Yaskawa INFORM job: AAA.JBI

/JOB
//NAME AAA
//POS
///NPOS 204,0,0,0,0,0
///TOOL 11
///POSTYPE PULSE
///PULSE
C00000=-67760,-23601,-34425,-10736,-67084,75715
C00001=-67760,-23601,-34425,-10736,-67084,75715
C00002=-69499,-30257,-42570,-18909,-69402,74527
C00003=-69664,-30877,-43349,-19628,-69583,74428
C00004=-69705,-31406,-44012,-20162,-69808,74223
C00005=-69657,-31867,-44586,-20565,-70063,73943
C00006=-69549,-32276,-45094,-20883,-70341,73613
C00007=-69400,-32646,-45556,-21151,-70634,73252
C00008=-69228,-32989,-45983,-21392,-70939,72872
C00009=-69041,-33312,-46388,-21624,-71251,72483
C00010=-68847,-33623,-46778,-21857,-71568,72091
C00011=-68651,-33924,-47158,-22097,-71886,71699
C00012=-68455,-34220,-47531,-22349,-72206,71309
C00013=-68258,-34512,-47898,-22611,-72524,70923
C00014=-68061,-34801,-48261,-22885,-72842,70541
C00015=-67864,-35088,-48619,-23168,-73158,70162
C00016=-67664,-35372,-48972,-23459,-73473,69786
C00017=-67462,-35653,-49319,-23757,-73786,69413
C00018=-67255,-35930,-49660,-24059,-74096,69042
C00019=-67043,-36203,-49993,-24363,-74405,68672
C00020=-66826,-36471,-50319,-24671,-74712,68304
C00021=-66603,-36736,-50637,-24979,-75016,67938
C00022=-66373,-36997,-50948,-25288,-75318,67573
C00023=-66137,-37255,-51251,-25599,-75616,67211
C00024=-65895,-37511,-51549,-25910,-75911,66851
C00025=-65647,-37765,-51840,-26222,-76201,66493
C00026=-65393,-38019,-52126,-26535,-76486,66139
C00027=-65133,-38273,-52409,-26849,-76767,65789
C00028=-64867,-38529,-52687,-27164,-77041,65442
C00029=-64596,-38787,-52963,-27481,-77309,65099
C00030=-64319,-39049,-53236,-27798,-77570,64761
C00031=-64036,-39314,-53506,-28117,-77824,64427
C00032=-63747,-39584,-53775,-28435,-78070,64097
C00033=-63453,-39857,-54041,-28754,-78309,63772
C00034=-63152,-40136,-54305,-29073,-78541,63450
C00035=-62844,-40418,-54566,-29390,-78765,63132
C00036=-62529,-40703,-54824,-29706,-78981,62818
C00037=-62206,-40991,-55077,-30019,-79190,62508
C00038=-61875,-41281,-55326,-30328,-79393,62200
C00039=-61536,-41572,-55568,-30634,-79589,61896
C00040=-61188,-41863,-55804,-30936,-79778,61593
C00041=-60831,-42153,-56033,-31232,-79961,61294
C00042=-60465,-42441,-56253,-31523,-80139,60996
C00043=-60089,-42725,-56464,-31808,-80311,60700
C00044=-59703,-43005,-56665,-32086,-80478,60405
C00045=-59307,-43279,-56855,-32357,-80640,60112
C00046=-58901,-43548,-57035,-32621,-80798,59821
C00047=-58485,-43810,-57203,-32878,-80951,59530
C00048=-58059,-44064,-57359,-33128,-81100,59241
C00049=-57623,-44310,-57503,-33370,-81246,58954
C00050=-57177,-44547,-57634,-33605,-81387,58667
C00051=-56721,-44775,-57753,-33832,-81525,58381
C00052=-56255,-44994,-57859,-34052,-81659,58097
C00053=-55780,-45203,-57953,-34264,-81790,57814
C00054=-55295,-45402,-58034,-34469,-81917,57533
C00055=-54801,-45591,-58102,-34667,-82040,57252
C00056=-54298,-45769,-58157,-34858,-82161,56973
C00057=-53786,-45937,-58199,-35042,-82278,56696
C00058=-53265,-46094,-58229,-35219,-82391,56420
C00059=-52736,-46240,-58247,-35389,-82502,56145
C00060=-52199,-46376,-58251,-35552,-82609,55872
C00061=-51653,-46500,-58244,-35709,-82714,55600
C00062=-51099,-46612,-58224,-35858,-82815,55330
C00063=-50537,-46714,-58191,-36001,-82914,55061
C00064=-49967,-46803,-58146,-36137,-83009,54795
C00065=-49390,-46881,-58088,-36267,-83102,54529
C00066=-48805,-46947,-58019,-36390,-83192,54265
C00067=-48213,-47001,-57937,-36507,-83280,54003
C00068=-47613,-47043,-57843,-36616,-83365,53743
C00069=-47007,-47072,-57737,-36720,-83448,53484
C00070=-46393,-47090,-57619,-36817,-83528,53227
C00071=-45773,-47096,-57489,-36907,-83606,52972
C00072=-45145,-47090,-57348,-36991,-83682,52718
C00073=-44512,-47072,-57195,-37068,-83755,52466
C00074=-43871,-47043,-57031,-37139,-83826,52216
C00075=-43225,-47002,-56855,-37204,-83895,51968
C00076=-42572,-46949,-56669,-37262,-83961,51722
C00077=-41913,-46886,-56472,-37313,-84026,51478
C00078=-41248,-46811,-56265,-37358,-84088,51235
C00079=-40577,-46725,-56047,-37396,-84148,50994
C00080=-39899,-46628,-55818,-37428,-84206,50756
C00081=-39216,-46520,-55579,-37453,-84262,50519
C00082=-38527,-46401,-55330,-37470,-84316,50284
C00083=-37832,-46270,-55070,-37481,-84369,50051
C00084=-37131,-46128,-54800,-37485,-84420,49819
C00085=-36423,-45974,-54518,-37481,-84469,49590
C00086=-35710,-45808,-54226,-37469,-84518,49362
C00087=-34991,-45630,-53923,-37450,-84566,49135
C00088=-34265,-45438,-53609,-37423,-84614,48911
C00089=-33534,-45233,-53282,-37387,-84661,48688
C00090=-32796,-45014,-52944,-37344,-84709,48466
C00091=-32052,-44781,-52594,-37291,-84757,48246
C00092=-31301,-44532,-52232,-37230,-84806,48027
C00093=-30544,-44269,-51857,-37160,-84857,47809
C00094=-29780,-43989,-51469,-37080,-84908,47593
C00095=-29010,-43694,-51068,-36991,-84962,47378
C00096=-28234,-43383,-50655,-36893,-85018,47165
C00097=-27450,-43055,-50228,-36785,-85075,46952
C00098=-26661,-42711,-49788,-36668,-85136,46741
C00099=-25864,-42351,-49335,-36540,-85199,46530
C00100=-25060,-41974,-48869,-36402,-85265,46321
C00101=-24250,-41581,-48391,-36254,-85333,46114
C00102=-23433,-41173,-47899,-36096,-85405,45907
C00103=-22609,-40749,-47396,-35927,-85479,45702
C00104=-21778,-40310,-46881,-35747,-85557,45497
C00105=-20940,-39856,-46354,-35556,-85638,45294
C00106=-20094,-39388,-45815,-35355,-85721,45093
C00107=-19241,-38906,-45265,-35142,-85808,44892
C00108=-18381,-38410,-44705,-34918,-85897,44693
C00109=-17513,-37901,-44133,-34682,-85990,44495
C00110=-16638,-37379,-43552,-34434,-86086,44298
C00111=-15755,-36843,-42960,-34174,-86186,44103
C00112=-14863,-36295,-42358,-33902,-86289,43909
C00113=-13964,-35733,-41745,-33617,-86395,43716
C00114=-13056,-35157,-41123,-33319,-86506,43524
C00115=-12139,-34568,-40490,-33008,-86622,43333
C00116=-11214,-33965,-39847,-32684,-86742,43143
C00117=-10280,-33347,-39194,-32346,-86867,42954
C00118=-9338,-32714,-38530,-31995,-86998,42766
C00119=-8386,-32066,-37856,-31629,-87135,42579
C00120=-7425,-31401,-37171,-31250,-87278,42392
C00121=-6454,-30721,-36476,-30856,-87429,42206
C00122=-5474,-30023,-35771,-30448,-87587,42021
C00123=-4485,-29308,-35055,-30026,-87753,41836
C00124=-3487,-28576,-34329,-29590,-87927,41652
C00125=-2479,-27827,-33594,-29139,-88109,41468
C00126=-1462,-27060,-32849,-28674,-88300,41285
C00127=-435,-26275,-32095,-28195,-88500,41102
C00128=600,-25474,-31333,-27702,-88709,40920
C00129=1645,-24655,-30563,-27196,-88928,40738
C00130=2698,-23819,-29786,-26676,-89155,40557
C00131=3760,-22967,-29004,-26143,-89393,40376
C00132=4829,-22099,-28216,-25597,-89639,40196
C00133=5907,-21215,-27423,-25040,-89895,40016
C00134=6992,-20316,-26627,-24470,-90160,39837
C00135=8084,-19401,-25829,-23890,-90435,39659
C00136=9182,-18472,-25028,-23298,-90719,39481
C00137=10286,-17527,-24227,-22697,-91013,39303
C00138=11396,-16568,-23425,-22087,-91317,39126
C00139=12510,-15594,-22623,-21469,-91631,38949
C00140=13627,-14604,-21823,-20844,-91954,38773
C00141=14748,-13600,-21024,-20213,-92288,38597
C00142=15870,-12581,-20228,-19576,-92632,38422
C00143=16993,-11546,-19434,-18936,-92987,38246
C00144=18117,-10495,-18644,-18292,-93352,38071
C00145=19239,-9428,-17858,-17648,-93728,37896
C00146=20359,-8345,-17076,-17003,-94115,37720
C00147=21476,-7246,-16299,-16360,-94513,37544
C00148=22589,-6130,-15528,-15719,-94922,37368
C00149=23696,-4998,-14762,-15082,-95343,37191
C00150=24796,-3848,-14001,-14451,-95774,37014
C00151=25888,-2681,-13246,-13826,-96216,36836
C00152=26971,-1496,-12498,-13210,-96670,36656
C00153=28044,-292,-11755,-12604,-97135,36476
C00154=29106,930,-11018,-12009,-97612,36294
C00155=30155,2171,-10286,-11426,-98100,36110
C00156=31190,3432,-9560,-10858,-98600,35925
C00157=32210,4713,-8838,-10304,-99112,35738
C00158=33215,6015,-8121,-9767,-99636,35548
C00159=34204,7338,-7408,-9248,-100171,35356
C00160=35174,8682,-6700,-8748,-100719,35160
C00161=36126,10048,-5995,-8268,-101279,34962
C00162=37059,11434,-5295,-7809,-101849,34761
C00163=37972,12840,-4598,-7372,-102430,34556
C00164=38864,14264,-3907,-6958,-103021,34348
C00165=39735,15705,-3222,-6567,-103621,34136
C00166=40585,17162,-2543,-6201,-104228,33920
C00167=41414,18631,-1872,-5858,-104841,33701
C00168=42221,20110,-1210,-5541,-105459,33478
C00169=43006,21596,-558,-5248,-106079,33251
C00170=43770,23088,82,-4980,-106701,33021
C00171=44512,24583,711,-4737,-107323,32787
C00172=45234,26079,1326,-4518,-107944,32550
C00173=45934,27576,1928,-4324,-108564,32309
C00174=46614,29074,2518,-4155,-109182,32065
C00175=47273,30571,3095,-4011,-109798,31817
C00176=47912,32069,3659,-3892,-110412,31565
C00177=48530,33569,4213,-3799,-111025,31308
C00178=49128,35070,4755,-3731,-111637,31047
C00179=49705,36574,5287,-3689,-112249,30781
C00180=50262,38079,5807,-3674,-112859,30510
C00181=50799,39584,6317,-3685,-113467,30234
C00182=51316,41089,6814,-3723,-114072,29952
C00183=51814,42589,7298,-3787,-114673,29665
C00184=52294,44083,7767,-3877,-115267,29373
C00185=52755,45568,8220,-3992,-115854,29077
C00186=53199,47042,8657,-4132,-116433,28776
C00187=53627,48504,9076,-4296,-117002,28470
C00188=54038,49954,9478,-4483,-117562,28160
C00189=54435,51394,9863,-4693,-118113,27846
C00190=54816,52823,10233,-4927,-118655,27526
C00191=55182,54241,10585,-5183,-119188,27202
C00192=55534,55645,10920,-5461,-119711,26873
C00193=55874,57028,11234,-5760,-120219,26541
C00194=56204,58383,11523,-6075,-120706,26208
C00195=56525,59701,11786,-6404,-121169,25876
C00196=56840,60977,12021,-6742,-121603,25546
C00197=57148,62218,12232,-7090,-122014,25218
C00198=57447,63448,12428,-7454,-122415,24887
C00199=57731,64701,12623,-7847,-122827,24544
C00200=57992,65992,12821,-8280,-123258,24185
C00201=58239,67231,12987,-8736,-123655,23826
C00202=58534,68041,12995,-9088,-123781,23559
C00203=61755,77652,13511,-13475,-125162,20533
//INST
///DATE 2023/04/06 12:39
///ATTR SC,RW
///GROUP1 RB1
NOP
MOVJ C00000 VJ=5.0
TIMER T=1.00
MOVJ C00001 VJ=1.0
TIMER T=0.10
MOVL C00002 V=400.0
MOVL C00003 V=400.0
MOVL C00004 V=400.0
MOVL C00005 V=400.0
MOVL C00006 V=400.0
MOVL C00007 V=400.0
MOVL C00008 V=400.0
MOVL C00009 V=400.0
MOVL C00010 V=400.0
MOVL C00011 V=400.0
MOVL C00012 V=400.0
MOVL C00013 V=400.0
MOVL C00014 V=400.0
MOVL C00015 V=400.0
MOVL C00016 V=400.0
MOVL C00017 V=400.0
MOVL C00018 V=400.0
MOVL C00019 V=400.0
MOVL C00020 V=400.0
MOVL C00021 V=400.0
MOVL C00022 V=400.0
MOVL C00023 V=400.0
MOVL C00024 V=400.0
MOVL C00025 V=400.0
MOVL C00026 V=400.0
MOVL C00027 V=400.0
MOVL C00028 V=400.0
MOVL C00029 V=400.0
MOVL C00030 V=400.0
MOVL C00031 V=400.0
MOVL C00032 V=400.0
MOVL C00033 V=400.0
MOVL C00034 V=400.0
MOVL C00035 V=400.0
MOVL C00036 V=400.0
MOVL C00037 V=400.0
MOVL C00038 V=400.0
MOVL C00039 V=400.0
MOVL C00040 V=400.0
MOVL C00041 V=400.0
MOVL C00042 V=400.0
MOVL C00043 V=400.0
MOVL C00044 V=400.0
MOVL C00045 V=400.0
MOVL C00046 V=400.0
MOVL C00047 V=400.0
MOVL C00048 V=400.0
MOVL C00049 V=400.0
MOVL C00050 V=400.0
MOVL C00051 V=400.0
MOVL C00052 V=400.0
MOVL C00053 V=400.0
MOVL C00054 V=400.0
MOVL C00055 V=400.0
MOVL C00056 V=400.0
MOVL C00057 V=400.0
MOVL C00058 V=400.0
MOVL C00059 V=400.0
MOVL C00060 V=400.0
MOVL C00061 V=400.0
MOVL C00062 V=400.0
MOVL C00063 V=400.0
MOVL C00064 V=400.0
MOVL C00065 V=400.0
MOVL C00066 V=400.0
MOVL C00067 V=400.0
MOVL C00068 V=400.0
MOVL C00069 V=400.0
MOVL C00070 V=400.0
MOVL C00071 V=400.0
MOVL C00072 V=400.0
MOVL C00073 V=400.0
MOVL C00074 V=400.0
MOVL C00075 V=400.0
MOVL C00076 V=400.0
MOVL C00077 V=400.0
MOVL C00078 V=400.0
MOVL C00079 V=400.0
MOVL C00080 V=400.0
MOVL C00081 V=400.0
MOVL C00082 V=400.0
MOVL C00083 V=400.0
MOVL C00084 V=400.0
MOVL C00085 V=400.0
MOVL C00086 V=400.0
MOVL C00087 V=400.0
MOVL C00088 V=400.0
MOVL C00089 V=400.0
MOVL C00090 V=400.0
MOVL C00091 V=400.0
MOVL C00092 V=400.0
MOVL C00093 V=400.0
MOVL C00094 V=400.0
MOVL C00095 V=400.0
MOVL C00096 V=400.0
MOVL C00097 V=400.0
MOVL C00098 V=400.0
MOVL C00099 V=400.0
MOVL C00100 V=400.0
MOVL C00101 V=400.0
MOVL C00102 V=400.0
MOVL C00103 V=400.0
MOVL C00104 V=400.0
MOVL C00105 V=400.0
MOVL C00106 V=400.0
MOVL C00107 V=400.0
MOVL C00108 V=400.0
MOVL C00109 V=400.0
MOVL C00110 V=400.0
MOVL C00111 V=400.0
MOVL C00112 V=400.0
MOVL C00113 V=400.0
MOVL C00114 V=400.0
MOVL C00115 V=400.0
MOVL C00116 V=400.0
MOVL C00117 V=400.0
MOVL C00118 V=400.0
MOVL C00119 V=400.0
MOVL C00120 V=400.0
MOVL C00121 V=400.0
MOVL C00122 V=400.0
MOVL C00123 V=400.0
MOVL C00124 V=400.0
MOVL C00125 V=400.0
MOVL C00126 V=400.0
MOVL C00127 V=400.0
MOVL C00128 V=400.0
MOVL C00129 V=400.0
MOVL C00130 V=400.0
MOVL C00131 V=400.0
MOVL C00132 V=400.0
MOVL C00133 V=400.0
MOVL C00134 V=400.0
MOVL C00135 V=400.0
MOVL C00136 V=400.0
MOVL C00137 V=400.0
MOVL C00138 V=400.0
MOVL C00139 V=400.0
MOVL C00140 V=400.0
MOVL C00141 V=400.0
MOVL C00142 V=400.0
MOVL C00143 V=400.0
MOVL C00144 V=400.0
MOVL C00145 V=400.0
MOVL C00146 V=400.0
MOVL C00147 V=400.0
MOVL C00148 V=400.0
MOVL C00149 V=400.0
MOVL C00150 V=400.0
MOVL C00151 V=400.0
MOVL C00152 V=400.0
MOVL C00153 V=400.0
MOVL C00154 V=400.0
MOVL C00155 V=400.0
MOVL C00156 V=400.0
MOVL C00157 V=400.0
MOVL C00158 V=400.0
MOVL C00159 V=400.0
MOVL C00160 V=400.0
MOVL C00161 V=400.0
MOVL C00162 V=400.0
MOVL C00163 V=400.0
MOVL C00164 V=400.0
MOVL C00165 V=400.0
MOVL C00166 V=400.0
MOVL C00167 V=400.0
MOVL C00168 V=400.0
MOVL C00169 V=400.0
MOVL C00170 V=400.0
MOVL C00171 V=400.0
MOVL C00172 V=400.0
MOVL C00173 V=400.0
MOVL C00174 V=400.0
MOVL C00175 V=400.0
MOVL C00176 V=400.0
MOVL C00177 V=400.0
MOVL C00178 V=400.0
MOVL C00179 V=400.0
MOVL C00180 V=400.0
MOVL C00181 V=400.0
MOVL C00182 V=400.0
MOVL C00183 V=400.0
MOVL C00184 V=400.0
MOVL C00185 V=400.0
MOVL C00186 V=400.0
MOVL C00187 V=400.0
MOVL C00188 V=400.0
MOVL C00189 V=400.0
MOVL C00190 V=400.0
MOVL C00191 V=400.0
MOVL C00192 V=400.0
MOVL C00193 V=400.0
MOVL C00194 V=400.0
MOVL C00195 V=400.0
MOVL C00196 V=400.0
MOVL C00197 V=400.0
MOVL C00198 V=400.0
MOVL C00199 V=400.0
MOVL C00200 V=400.0
MOVL C00201 V=400.0
MOVL C00202 V=400.0
MOVL C00203 V=400.0
END
